// TIA Portal V17 export
// export: Created 2024-08-07T21:44:10.9878196Z, ExportSetting WithDefaults, DisplayName Totally Integrated Automation Portal, DisplayVersion V17 Update 7, DisplayName TIA Portal Openness, DisplayVersion V17 Update 7, DisplayName TIA Portal Version Control Interface, DisplayVersion V17, DisplayName SINAMICS Startdrive Advanced, DisplayVersion V17 SP2, DisplayName SINAMICS Startdrive G110M, G120, G120C, G120D, G120P, G115D, DisplayVersion V17 SP2, DisplayName SINAMICS Startdrive G130, G150, S120, S150, SINAMICS MV, S210, DisplayVersion V17 SP2, DisplayName STEP 7 Professional, DisplayVersion V17 Update 7, DisplayName STEP 7 Safety, DisplayVersion V17 Update 6, DisplayName WinCC Advanced / Unified PC, DisplayVersion V17 Update 7
FUNCTION_BLOCK "6. Call_M004_NTRS"   // FB2006, LAD
{ S7_Optimized_Access := 'TRUE' }
VERSION : 0.1
// stored: AutoNumber false, IsIECCheckEnabled false, IsRetainMemResEnabled false, MemoryReserve 100, SetENOAutomatically false, UDAEnableTagReadback false
   VAR_INPUT
      nTRSTag : Bool;
   END_VAR
   VAR
      nTRSTagTemp : Bool;
   END_VAR
BEGIN

REGION Network 1 (SCL)
   IF #nTRSTag <> #nTRSTagTemp THEN

       "MII_Interface_Data".MII_METHODS.M004_NTRS.Inputs.PLC_ID := "MII_Parameters".Connection.PLC_ID;
       "MII_Interface_Data".MII_METHODS.M004_NTRS.Inputs.PLANT := "MII_Parameters".Connection.PlantID;
       "MII_Interface_Data".MII_METHODS.M004_NTRS.Inputs.STOPPAGE := #nTRSTag;
       "MII_Interface_Data".MII_METHODS.M004_NTRS.Inputs.CAUSE := WSTRING#'1S014040';
       //Call the method 
       "1. DMC_setConnection_DB".CallBuffer[6] := TRUE;

       #nTRSTagTemp := #nTRSTag;
   END_IF;
END_REGION
END_FUNCTION_BLOCK
